{attribute 'qualified_only'}
VAR_GLOBAL
END_VAR

(* stored: Version 1.1.0.1, ProductVersion 3.1.4024.12
   GVL G_Task2: Id {f5ec6e46-21cf-4f28-8d49-89ffe42e4084} *)
